TYPE ST_InsulationMonitor_params :
STRUCT
	i_EarthSystemDetectionDelay		:INT := 60; // Seconds
END_STRUCT
END_TYPE

(* stored: Version 1.1.0.1, ProductVersion 3.1.4026.18
   DUT ST_InsulationMonitor_params: Id {b22150b5-56ab-46a6-bdba-ef3613966293} *)
